(* IEC 61131-3 sources: lacyccom-procedural/src/drive_functions/blocks (part 3) *)

(* ---- LAcycCom_DriveRamToRom.st ---- *)
USING System.Timer;
USING Siemens.Simatic.DistributedIO;

NAMESPACE Simatic.Ax.LAcycCom.Procedural
  TYPE INTERNAL
    LAcycCom_DriveRamToRomStates : SINT (
      FB_IDLE := SINT#0,   // Idle state in FB
      FB_FIRST_CYCLE := SINT#1,   // First cycle state in FB
      FB_ALLOCATE := SINT#2,   // Allocating a buffer element in request buffer DB
      FB_GET_RESOURCE := SINT#3,   // State to check if the communication to the drive object can be established
      FB_BUSY := SINT#4,   // Busy state in FB
      FB_RELEASE := SINT#5,   // State to return the allocated index
      FB_DONE := SINT#6,   // Done state in FB
      FB_ERROR := SINT#7,   // Error state in FB
      FB_BUSY_READ := SINT#8,   // State of configuration drive object data (read parameter r3996)
      FB_BUSY_WriteRecord_READ := SINT#9,   // WriteRecord in busy state
      FB_BUSY_ReadRecord_READ := SINT#10,   // ReadRecord in busy state
      FB_BUSY_WRITE_PARAM_971 := SINT#11,   // State of configuration drive object data (write parameter p971)
      FB_BUSY_WriteRecord_WRITE_PARAM_971 := SINT#12,   // WriteRecord in busy state
      FB_BUSY_ReadRecord_WRITE_PARAM_971 := SINT#13,   // ReadRecord in busy state
      FB_BUSY_WRITE_PARAM_977 := SINT#14,   // State of configuration drive object data (write parameter p977)
      FB_BUSY_WriteRecord_WRITE_PARAM_977 := SINT#15,   // WriteRecord in busy state
      FB_BUSY_ReadRecord_WRITE_PARAM_977 := SINT#16,   // ReadRecord in busy state
      FB_BUSY_CYCLE_TIMER := SINT#17,   // Cyclic OnDelay in busy state
      FB_BUSY_CHECK_PARAM_971 := SINT#18,   // State of configuration drive object data (read parameter r3996)
      FB_BUSY_WriteRecord_CHECK_971 := SINT#19,   // WriteRecord in busy state
      FB_BUSY_ReadRecord_CHECK_971 := SINT#20,   // ReadRecord in busy state
      FB_BUSY_CHECK_PARAM_977 := SINT#21,   // State of configuration drive object data (read parameter p977)
      FB_BUSY_WriteRecord_CHECK_977 := SINT#22,   // WriteRecord in busy state
      FB_BUSY_ReadRecord_CHECK_977 := SINT#23,   // ReadRecord in busy state
      FB_BUSY_CHECK_PROGRESS := SINT#24,   // Check RAM to ROM progress
      FB_BUSY_WAIT := SINT#25   // State when temporary error occurred
    ) := FB_IDLE;
  END_TYPE

  ///------------------------------------------------------------------------------------------
  /// SIEMENS AG
	/// (c)Copyright 2026 All Rights Reserved
	///------------------------------------------------------------------------------------------
	/// Library: LAcycCom
	/// Tested with: S7-1513-1 PN
	/// Engineering: SIMATIC AX
	/// Restrictions: ---
	/// Requirements: S7-1200 / S7-1500
	///               FB LAcycCom_ResourceManager is required
	/// Functionality: Copy RAM to ROM of a specific drive object.
  ///------------------------------------------------------------------------------------------
  FUNCTION_BLOCK LAcycCom_DriveRamToRom
    {S7.Extern = ReadWrite}
    VAR_INPUT
      execute : BOOL;   /// TRUE: Rising edge starts the functionality once
      driveObjectId : INT := -1;   /// Optional: Identification number of the drive object (value <0: driveObjectId is not used, i.e. the corresponding drive object is only addressed via the hardwareId)
      hardwareId : UINT;   /// Hardware identifier of the hardware module
      enableSavingOfWholeDriveSystem : BOOL;   /// TRUE: Enable saving of all parameters of all drive objects of a multi drive system (e.g. S120). Note: parameter p977 must therefore be available at the addressed drive object. If p977 is not available p971 is written, i.e., the setting also works for single drive systems (e.g. G120)
    END_VAR

    {S7.Extern = ReadOnly}
    VAR_OUTPUT
      done : BOOL;   /// TRUE: RAM data successfully written to ROM
      busy : BOOL;   /// TRUE: FB is not finished and new output values can be expected
      error : BOOL;   /// TRUE: Rising edge informs that an error occurred during the execution of the FB
      status : LAcycCom_DriveFunctionStatus := LAcycCom_DriveFunctionStatus#STATUS_NO_CALL;   /// Status identifier
      diagnostics : LAcycCom_typeDriveDiagnostics;   /// Diagnostics structure
    END_VAR

    VAR_IN_OUT
      requestBufferHeader : LAcycCom_typeRequestBufferHeader;   /// Interface for header of request buffer
      requestBuffer : ARRAY[*] OF LAcycCom_typeRequestBufferElement;   /// Interface for request buffer
    END_VAR

    VAR
      _busy : BOOL := FALSE;   /// Static value for output busy
      _done : BOOL := FALSE;   /// Static value for output done
      _error : BOOL := FALSE;   /// Static value for output error
      _executeOld : BOOL := FALSE;   /// Old value of execute for edge detection
      _cmdBusy : BOOL := FALSE;   /// TRUE: Process is not yet complete
      _cmdDone : BOOL := FALSE;   /// TRUE: Data record was transferred
      _cmdError : BOOL := FALSE;   /// TRUE: An error occurred during processing
      _timerStart : BOOL := FALSE;   /// TRUE: Starts OnDelay
      _refNo : BYTE := BYTE#16#00;   /// Reference number of request
      _doId : BYTE := BYTE#16#00;   /// Intern identification number of the drive object
      _status : LAcycCom_DriveFunctionStatus := LAcycCom_DriveFunctionStatus#STATUS_NO_CALL;   /// Static value for output status
      _subfunctionStatus : WORD := WORD#16#0000;   /// Block status or error information
      _withoutResourceManager : BOOL := FALSE;   /// TRUE: No resource manager available; FALSE: Resource manager available
      _stateNumber : SINT := SINT#0;   /// State of the FB when error occurred
      _fbState : SINT := LAcycCom_DriveRamToRomStates#FB_IDLE;   /// States in the function block state machine
      _fbSubState : SINT := LAcycCom_DriveRamToRomStates#FB_BUSY_WriteRecord_WRITE_PARAM_971;   /// States in the function block during processing (busy state)
      _fbSubStateOld : SINT := LAcycCom_DriveRamToRomStates#FB_BUSY_WriteRecord_WRITE_PARAM_971;   /// Previous state when temporary error occurs
      _errorCount : UInt := UINT#0;   /// Error counter of retry request
      _allocatedIndex : INT := 0;   /// Allocated element index in the buffer DB
      _countOfElements : INT := 0;   /// Number of parameters in the dataset
      _firstParameterError : INT := -1;   /// Number of parameter at which the error occurred (-1: no parameter with error)
      _hwId : UINT := UINT#0;   /// Intern hardware identifier of the hardware module
      _warningRetriggering : BOOL;   /// TRUE: Input execute is set during processing
      _dataRecordNo : DINT;   /// Used data record
      _cyclicTimerStart : BOOL;   /// TRUE: Starts the OnDelay
      _parameter : ARRAY[0..NO_OF_PARAMETERS_UPPER_LIM] OF LAcycCom_typeParameter;   /// Parameter dataset
      _parameterRam2Rom : ARRAY[0..0] of LAcycCom_typeParameter;   /// Parameter dataset for write Ram2Rom
      _reqWriteParameterHeader : LAcycCom_typeParameterHeader;   /// Request telegram to change the parameter values
      _reqWriteParameterData : ARRAY[0..LENGTH_WRITE_PARAMETER_TELEGRAM_UPPER_LIM] OF BYTE;   /// List of parameter (max. 16 parameter)
      _reqReadParameterHeader : LAcycCom_typeParameterHeader;   /// Request telegram
      _reqReadParameterAddress : ARRAY[0..NO_OF_PARAMETERS_UPPER_LIM] OF LAcycCom_typeParameterAddress;   /// Parameter data in telegram
      _respParameterHeader : LAcycCom_typeParameterHeader;   /// Response telegram
      _respParameterData : ARRAY[0..LENGTH_READ_PARAMETER_TELEGRAM_UPPER_LIM] OF BYTE;   /// List of parameter (max. 16 parameter)
      _reqReadParameterInit : LAcycCom_typeParameterAddress := ( attribute := BYTE#16#10, elementNo := BYTE#16#01, parameterNo := UINT#0, index := UINT#0 );   /// Initialisation of the parameter dataset
      _instWriteRecord  : WriteRecord;   /// WriteRecord command
      _instReadRecord : ReadRecord;   /// ReadRecord command
      _instOnDelay : OnDelay;   /// OnDelay
    END_VAR

    VAR_TEMP
      tempCmdValid : BOOL;   // TRUE: New data record was received and is valid
      tempIndex : INT;   // Temporary loop index variable
      tempLastQueueElement : INT;   // Last element in queue
      tempPointer : INT;   // Temporary pointer variable
      tempWord : WORD;   // Temporary word variable
      tempUDint : UDINT;   // Temporary udint variable
      tempStatusWord : WORD;   // Temporary status
      tempCmdStatus : DWORD;   // Temporary status of WriteRecord and ReadRecord command
      tempVoidDiagnostics : LAcycCom_typeDriveDiagnostics;   // Temporary empty diagnostics structure
      tempVoidHeader : LAcycCom_typeParameterHeader;   // Temporary empty header structure
      tempRecord : ARRAY[0..239] OF BYTE;   // Temporary record buffer for WriteRecord and ReadRecord instruction
    END_VAR

    VAR CONSTANT
      MAX_ERROR_COUNT : UINT := UINT#40;   // Maximum error counter
      NO_OF_PARAMETERS_UPPER_LIM : INT := 1;   // Maximum count of parameters
      LENGTH_WRITE_PARAMETER_TELEGRAM_UPPER_LIM : INT := 23;   // Maximum length of write telegram in Byte
      LENGTH_READ_PARAMETER_TELEGRAM_UPPER_LIM : INT := 11;   // Maximum length of read telegram in Byte
      ALL_ELEMENTS_OCCUPIED : INT := -1;   // All buffer elements are occupied
      TIMER_ALLOCATION : TIME := T#10S;   // Timer limit for allocating a buffer element
      TIMER_TEMP_ERROR : TIME := T#200MS;   // Waiting time until next system function block call
      TIMER_CYCLIC : TIME := T#500MS;   // Timer interval of checking the result of the Ram to Rom process
      MAX_DRIVE_OBJECT_NO : INT := 254;   // Maximum drive object number limited by SINAMICS p101
    END_VAR

    // Check if FB is triggered
    IF (execute = TRUE) AND (_executeOld = FALSE) AND (_busy = TRUE) THEN
      // Input execute is set during processing
      _status := LAcycCom_DriveFunctionStatus#WARN_EXECUTE_SET_DURING_PROCESSING;
      _warningRetriggering := TRUE;
      _executeOld := execute;

    ELSIF (execute = TRUE) AND (_executeOld = FALSE) THEN
      // First call
      // Initialisation
      _done := FALSE;
      _error := FALSE;
      //_status := LAcycCom_DriveFunctionStatus#STATUS_FIRST_CALL;
      _allocatedIndex := 0;
      _hwId := UINT#0;
      _subfunctionStatus := WORD#16#0;
      _doId := BYTE#0;
      _dataRecordNo := 0;
      _stateNumber := SINT#0;
      _firstParameterError := -1;
      _cmdBusy := FALSE;
      _cmdDone := FALSE;
      _cmdError := FALSE;
      _errorCount := UINT#0;
      _countOfElements := 0;
      _warningRetriggering := FALSE;
      _fBSubState := LAcycCom_DriveRamToRomStates#FB_BUSY_READ;
      _fBState := LAcycCom_DriveRamToRomStates#FB_FIRST_CYCLE;

      // Initialize functionality after triggering FB, e.g. reset of values
      //-----------------------------------------------------------------------------------
      _instOnDelay(signal := FALSE,
              duration := TIMER_ALLOCATION);

      // Functionality is busy
      _busy := TRUE;

      // Reset other outputs
      _error := FALSE;
      //_status := LAcycCom_DriveFunctionStatus#STATUS_FIRST_CALL;

      busy := _busy;
      error := _error;
      _executeOld := execute;
      RETURN;

      // FB is currently inactive
    ELSIF (execute = FALSE) AND (_busy = FALSE) AND
        (_error = TRUE OR _done = TRUE)
    THEN
      _error := FALSE;
      _busy := FALSE;
      _done := FALSE;
      _fBState := LAcycCom_DriveRamToRomStates#FB_IDLE;

      // Write outputs
      _status := LAcycCom_DriveFunctionStatus#STATUS_NO_CALL;
      busy := _busy;
      done := _done;
      error := _error;

      _executeOld := execute;
      RETURN;

      // FB is currently executed and not finished
    ELSIF _busy = TRUE THEN
      _executeOld := execute;

      // FB finished request
    ELSE
      _executeOld := execute;
      RETURN; //Wait for start of functionality
    END_IF;
    //----------------------------------------------------------------------------------------------

    IF (_busy = TRUE) AND (_error = FALSE) THEN  // Functionality running
        CASE _fBState OF
            LAcycCom_typeDriveActDeactStates#FB_FIRST_CYCLE:  // First cycle state

            // Clearing the sending reading buffer
            _reqReadParameterHeader := tempVoidHeader;
            _reqReadParameterAddress[0] := _reqReadParameterInit;

            // Clearing the sending write buffer
            _reqWriteParameterHeader := tempVoidHeader;
            FOR tempIndex := 0 TO LENGTH_WRITE_PARAMETER_TELEGRAM_UPPER_LIM DO
            _reqWriteParameterData[tempIndex] := BYTE#16#00;
            END_FOR;

            // Clearing the receive buffer
            _respParameterHeader := tempVoidHeader;
            FOR tempIndex := 0 TO LENGTH_READ_PARAMETER_TELEGRAM_UPPER_LIM DO
            _respParameterData[tempIndex] := BYTE#16#00;
            END_FOR;

            // Initialization after start
            IF driveObjectId < 0 THEN // V1.5
            _dataRecordNo := 16#B02E; // Base Mode Parameter Access local; doId not relevant
            _doId := BYTE#0;

            ELSIF (driveObjectId <= MAX_DRIVE_OBJECT_NO)
            AND (driveObjectId <> 0)
            THEN // V1.5.2
            _dataRecordNo := 47; // Data record 47; Base Mode Parameter Access global
            _doId := TO_BYTE(driveObjectId);

            ELSE // V1.5.2
            // Wrong drive object ID at input
            _error := TRUE;
            _stateNumber := _fBState;
            _status := LAcycCom_DriveFunctionStatus#ERR_INVALID_DRIVE_OBJECT_ID;
            _fBState := LAcycCom_typeDriveActDeactStates#FB_ERROR;
            END_IF;

            _hwId := hardwareId;
            diagnostics := tempVoidDiagnostics;
            diagnostics.driveObjectId := TO_SINT(_doId);
            diagnostics.hardwareId := _hwId;
            diagnostics.parameterCount := 2;
            _countOfElements := 2;
            diagnostics.firstParameterError := _firstParameterError; // V1.3.2
            diagnostics.errorValue := BYTE#16#FF; // V1.3.2

            _parameter[0].parameterNo := UINT#0;
            _parameter[1].parameterNo := UINT#0;
            _parameterRam2Rom[0].parameterNo := UINT#0; // V1.3.3

            _parameter[0].index := UINT#0;
            _parameter[1].index := UINT#0;
            _parameterRam2Rom[0].index := UINT#0;

            _parameter[0].realValue := REAL#0.0;
            _parameter[1].realValue := REAL#0.0;
            _parameterRam2Rom[0].realValue := REAL#0.0;

            _parameter[0].format := BYTE#16#00;
            _parameter[1].format := BYTE#16#00;
            _parameterRam2Rom[0].format := BYTE#16#00;

            _parameter[0].errorValue := BYTE#16#00;
            _parameter[1].errorValue := BYTE#16#00;
            _parameterRam2Rom[0].errorValue := BYTE#16#00;

            // Next state is depending on the FB mode
            IF (_withoutResourceManager = FALSE) AND (_error = FALSE) THEN
            _status := LAcycCom_DriveFunctionStatus#STATUS_ALLOCATE;
            _fBState := LAcycCom_typeDriveActDeactStates#FB_ALLOCATE;

            ELSIF (_withoutResourceManager = TRUE) AND (_error = FALSE) THEN
            _status := LAcycCom_DriveFunctionStatus#STATUS_BUSY;
            _fBState := LAcycCom_typeDriveActDeactStates#FB_BUSY;
            _fBSubState := LAcycCom_DriveRamToRomStates#FB_BUSY_READ;
            END_IF;

            LAcycCom_typeDriveActDeactStates#FB_ALLOCATE:
            // Allocation of a buffer element
            IF (requestBufferHeader.lockBuffer = FALSE) AND (requestBufferHeader.nextFreeElement >= requestBufferHeader.bufferLowerBound) AND (requestBufferHeader.nextFreeElement <= requestBufferHeader.bufferUpperBound) THEN
            requestBufferHeader.lockBuffer := TRUE;
            _allocatedIndex := requestBufferHeader.nextFreeElement;
            requestBuffer[_allocatedIndex].state := BYTE#16#00;
            requestBuffer[_allocatedIndex].state.%X0 := TRUE;
            requestBuffer[_allocatedIndex].hardwareId := _hwId;
            requestBuffer[_allocatedIndex].queueElementNext := -1;
            _timerStart := FALSE;
            _status := LAcycCom_DriveFunctionStatus#STATUS_GET_RESOURCE;
            _fBState := LAcycCom_typeDriveActDeactStates#FB_GET_RESOURCE;

            // Build up queue
            IF (requestBufferHeader.firstQueueElement >= 0) THEN
                // Find last queue element
                tempIndex := requestBufferHeader.firstQueueElement;
                WHILE (tempIndex >= 0) DO
                tempLastQueueElement := tempIndex;
                tempIndex := requestBuffer[tempIndex].queueElementNext;
                END_WHILE;

                // Insert into list after last element
                requestBuffer[tempLastQueueElement].queueElementNext := _allocatedIndex;
                requestBuffer[_allocatedIndex].queueElementPrevious := tempLastQueueElement;

            ELSE
                // Element is first element in queue
                requestBufferHeader.firstQueueElement := _allocatedIndex;
                requestBuffer[_allocatedIndex].queueElementPrevious := -1;
            END_IF;

            // Searching for the next free buffer element
            FOR tempIndex := requestBufferHeader.bufferLowerBound TO TO_INT(requestBufferHeader.bufferUpperBound) DO
                IF (requestBuffer[tempIndex].state.%X0 = FALSE) THEN
                requestBufferHeader.nextFreeElement := tempIndex;
                EXIT;
                END_IF;

                // All buffer elements are occupied
                IF (tempIndex = requestBufferHeader.bufferUpperBound) THEN
                requestBufferHeader.nextFreeElement := ALL_ELEMENTS_OCCUPIED;
                END_IF;
            END_FOR;

            requestBufferHeader.lockBuffer := FALSE;

            ELSIF (_instOnDelay.output = TRUE) THEN
            _error := TRUE;
            _stateNumber := _fBState;
            _status := LAcycCom_DriveFunctionStatus#ERR_ALLOCATION_TIME;
            _fBState := LAcycCom_typeDriveActDeactStates#FB_ERROR;

            ELSE
            ; // Waiting until lockbit is reset and a buffer element is available
            END_IF; // (#buffer.lockBuffer = FALSE) AND (#buffer.actualWriteIndex >= 0)

            _instOnDelay(signal := _timerStart,
                    duration := TIMER_ALLOCATION);

            _timerStart := TRUE;
            IF (_instOnDelay.output = TRUE) THEN
            _timerStart := FALSE;
            END_IF;

            LAcycCom_typeDriveActDeactStates#FB_GET_RESOURCE:

            // Check buffer index for correctness
            IF (_allocatedIndex < requestBufferHeader.bufferLowerBound) OR (_allocatedIndex > requestBufferHeader.bufferUpperBound) THEN
            _error := TRUE;
            _stateNumber := _fBState;
            _status := LAcycCom_DriveFunctionStatus#ERR_INVALID_BUF_INDEX;
            _fBState := LAcycCom_typeDriveActDeactStates#FB_ERROR;

            ELSE
            IF (requestBuffer[_allocatedIndex].state.%X0 = FALSE) OR
                (requestBuffer[_allocatedIndex].state.%X3 = TRUE)
            THEN
                // Request was rejected by buffer manager
                _error := TRUE;
                _stateNumber := _fBState;
                _status := LAcycCom_DriveFunctionStatus#ERR_REQUEST_REJECTED;
                _fBState := LAcycCom_typeDriveActDeactStates#FB_ERROR;

            ELSIF (requestBuffer[_allocatedIndex].state.%X2 = TRUE) THEN
                // Request already released
                _error := TRUE;
                _stateNumber := _fBState;
                _status := LAcycCom_DriveFunctionStatus#ERR_RESOURCE_RELEASED;
                _fBState := LAcycCom_typeDriveActDeactStates#FB_ERROR;

            ELSIF (requestBuffer[_allocatedIndex].state.%X1 = TRUE) THEN
                // Element is enabled
                _status := LAcycCom_DriveFunctionStatus#STATUS_BUSY;
                _fBState := LAcycCom_typeDriveActDeactStates#FB_BUSY;
                _fBSubState := LAcycCom_DriveRamToRomStates#FB_BUSY_READ;

            ELSE
                // Element not enabled yet
                //
                _status := LAcycCom_DriveFunctionStatus#STATUS_GET_RESOURCE;
            END_IF;

            END_IF;

            LAcycCom_typeDriveActDeactStates#FB_BUSY:

            IF ((requestBuffer[_allocatedIndex].state.%X1 = TRUE) AND (_withoutResourceManager = FALSE) AND ((requestBuffer[_allocatedIndex].state.%X3 = FALSE))) OR
            (_withoutResourceManager = TRUE)
            THEN

            CASE _fBSubState OF

                LAcycCom_DriveRamToRomStates#FB_BUSY_READ:
                // Creating header data
                _refNo := TO_BYTE(TO_SINT(_refNo) + 1);
                _reqReadParameterHeader.refNo := _refNo; // Telegram reference number
                _reqReadParameterHeader.reqId := BYTE#16#01;  // 0x01 = request parameters
                _reqReadParameterHeader.doId := _doId;  // Drive object identification number
                _reqReadParameterHeader.parameterNo := TO_BYTE(_countOfElements);  // Count of parameters

                // Copying the dataset into a static variable (depending on the used PLC data type)
                _parameter[0].index := UINT#0;
                _parameter[0].parameterNo := UINT#971; // Save drive object parameters
                _parameter[0].format := TO_BYTE(LAcycCom_DriveValueFormats#FORMAT_UNSIGNED_16);
                _parameter[1].index := UINT#0;
                _parameter[1].parameterNo := UINT#977; // Save all parameters
                _parameter[1].format := TO_BYTE(LAcycCom_DriveValueFormats#FORMAT_UNSIGNED_16);

                _reqReadParameterAddress[0].attribute := BYTE#16#10; // Attribute of parameters (0x10=Value, 0x30=Text)
                _reqReadParameterAddress[0].elementNo := BYTE#16#01; // No. of elements (for single elements=1)

                _reqReadParameterAddress[1].attribute := BYTE#16#10; // Attribute of parameters (0x10=Value, 0x30=Text)
                _reqReadParameterAddress[1].elementNo := BYTE#16#01; // No. of elements (for single elements=1)

                // Parameter number
                _reqReadParameterAddress[0].parameterNo := _parameter[0].parameterNo;
                _reqReadParameterAddress[1].parameterNo := _parameter[1].parameterNo;

                // Subindex of parameter
                _reqReadParameterAddress[0].index := _parameter[0].index;
                _reqReadParameterAddress[1].index := _parameter[1].index;

                _status := LAcycCom_DriveFunctionStatus#STATUS_BUSY;
                _fBState := LAcycCom_typeDriveActDeactStates#FB_BUSY;
                _fBSubState := LAcycCom_DriveRamToRomStates#FB_BUSY_WriteRecord_READ;

                LAcycCom_DriveRamToRomStates#FB_BUSY_WRITE_PARAM_971, LAcycCom_DriveRamToRomStates#FB_BUSY_WRITE_PARAM_977:

                // Initialize diagnostics and count of elements
                diagnostics.parameterCount := 1;
                _countOfElements := 1;

                // Clearing the receive buffer V1.3.3
                _respParameterHeader := tempVoidHeader;
                FOR tempIndex := 0 TO LENGTH_READ_PARAMETER_TELEGRAM_UPPER_LIM DO
                    _respParameterData[tempIndex] := BYTE#16#00;
                END_FOR;

                // Creating header data
                _refNo := TO_BYTE(TO_SINT(_refNo) + 1);
                _reqWriteParameterHeader.refNo := _refNo; // Telegram reference number
                _reqWriteParameterHeader.reqId := BYTE#16#02;  // 0x02 = change parameters
                _reqWriteParameterHeader.doId := _doId;  // Drive object identification number of CU
                _reqWriteParameterHeader.parameterNo := TO_BYTE(_countOfElements);  // Count of parameters

                // Copying the dataset into a static variable
                _parameterRam2Rom[0].index := UINT#0;
                IF (_fBSubState = LAcycCom_DriveRamToRomStates#FB_BUSY_WRITE_PARAM_971) THEN // V1.3.3
                    _parameterRam2Rom[0].parameterNo := UINT#971; // Save drive object parameters
                    _fBSubState := LAcycCom_DriveRamToRomStates#FB_BUSY_WriteRecord_WRITE_PARAM_971;
                ELSE
                    _parameterRam2Rom[0].parameterNo := UINT#977; // Save all parameters
                    _fBSubState := LAcycCom_DriveRamToRomStates#FB_BUSY_WriteRecord_WRITE_PARAM_977;
                END_IF;

                _parameterRam2Rom[0].format := TO_BYTE(LAcycCom_DriveValueFormats#FORMAT_UNSIGNED_16);
                _parameterRam2Rom[0].realValue := REAL#1.0;

                // Write parameter address
                _reqWriteParameterData[0] := BYTE#16#10; // Attribute of parameters (0x10=Value, 0x30=Text)
                _reqWriteParameterData[1] := BYTE#16#01; // No. of elements (for single elements=1)

                // Parameter number
                _reqWriteParameterData[2] := _parameterRam2Rom[0].parameterNo.%B1;
                _reqWriteParameterData[3] := _parameterRam2Rom[0].parameterNo.%B0;

                // Subindex of parameter
                _reqWriteParameterData[4] := _parameterRam2Rom[0].index.%B1;
                _reqWriteParameterData[5] := _parameterRam2Rom[0].index.%B0;

                _reqWriteParameterData[6] := _parameterRam2Rom[0].format; // Format of parameter
                _reqWriteParameterData[7] := BYTE#16#01; // Count of values

                // Parameter value (= 1.0)
                _reqWriteParameterData[8] := BYTE#16#00;
                _reqWriteParameterData[9] := BYTE#16#01;

                _status := LAcycCom_DriveFunctionStatus#STATUS_BUSY;
                _fBState := LAcycCom_typeDriveActDeactStates#FB_BUSY;

                LAcycCom_DriveRamToRomStates#FB_BUSY_CYCLE_TIMER:

                // Start cyclic timer
                _instOnDelay(signal := _cyclicTimerStart,
                              duration := TIMER_CYCLIC);

                _cyclicTimerStart := TRUE;
                IF (_instOnDelay.output = TRUE) THEN
                    _cyclicTimerStart := FALSE;
                    _fBSubState := _fBSubStateOld; // V1.3.3
                END_IF;

                LAcycCom_DriveRamToRomStates#FB_BUSY_CHECK_PARAM_971, LAcycCom_DriveRamToRomStates#FB_BUSY_CHECK_PARAM_977:

                // Clearing the receive buffer V1.3.3
                _respParameterHeader := tempVoidHeader;
                FOR tempIndex := 0 TO LENGTH_READ_PARAMETER_TELEGRAM_UPPER_LIM DO
                    _respParameterData[tempIndex] := BYTE#16#00;
                END_FOR;

                // Creating header data
                _refNo := TO_BYTE(TO_SINT(_refNo) + 1);
                _reqReadParameterHeader.refNo := _refNo; // Telegram reference number
                _reqReadParameterHeader.reqId := BYTE#16#01;  // 0x01 = request parameters
                _reqReadParameterHeader.doId := _doId;  // Drive object identification number of CU
                _reqReadParameterHeader.parameterNo := TO_BYTE(_countOfElements);  // Count of parameters

                IF _fBSubState = LAcycCom_DriveRamToRomStates#FB_BUSY_CHECK_PARAM_971 THEN // V1.3.3
                    _parameterRam2Rom[0].parameterNo := UINT#971; // Save drive object parameters
                    _fBSubState := LAcycCom_DriveRamToRomStates#FB_BUSY_WriteRecord_CHECK_971;

                ELSE
                    _parameterRam2Rom[0].parameterNo := UINT#977; // Save all parameters
                    _fBSubState := LAcycCom_DriveRamToRomStates#FB_BUSY_WriteRecord_CHECK_977;
                END_IF;

                _parameterRam2Rom[0].format := TO_BYTE(LAcycCom_DriveValueFormats#FORMAT_UNSIGNED_16);

                _status := LAcycCom_DriveFunctionStatus#STATUS_BUSY;
                _fBState := LAcycCom_typeDriveActDeactStates#FB_BUSY;

                // Copying the dataset into a static variable (depending on the used PLC data type)
                _parameterRam2Rom[0].index := UINT#0;

                _reqReadParameterAddress[0].attribute := BYTE#16#10; // Attribute of parameters (0x10=Value, 0x30=Text)
                _reqReadParameterAddress[0].elementNo := BYTE#16#01; // No. of elements (for single elements=1)

                // Parameter number
                _reqReadParameterAddress[0].parameterNo := _parameterRam2Rom[0].parameterNo;

                // Subindex of parameter
                _reqReadParameterAddress[0].index := _parameterRam2Rom[0].index;

                LAcycCom_DriveRamToRomStates#FB_BUSY_CHECK_PROGRESS:

                IF (_parameterRam2Rom[0].realValue = REAL#0.0) // Ram2Rom is completed
                THEN

                    // Next state is depending on the FB mode
                    IF (_withoutResourceManager = FALSE) AND (_error = FALSE) THEN
                    _status := LAcycCom_DriveFunctionStatus#STATUS_RELEASE;
                    _fBState := LAcycCom_typeDriveActDeactStates#FB_RELEASE;

                    ELSIF (_withoutResourceManager = TRUE) AND (_error = FALSE) THEN
                    _status := LAcycCom_DriveFunctionStatus#STATUS_EXECUTION_FINISHED;
                    _fBState := LAcycCom_typeDriveActDeactStates#FB_DONE;
                    END_IF; // _mode = #MODE_WITH_BUFFER_MANAGER

                ELSE
                    _status := LAcycCom_DriveFunctionStatus#STATUS_BUSY;
                    _fBSubState := LAcycCom_DriveRamToRomStates#FB_BUSY_CYCLE_TIMER;
                END_IF;

                // Writing the dataset configuration into the drive object
                LAcycCom_DriveRamToRomStates#FB_BUSY_WriteRecord_READ, LAcycCom_DriveRamToRomStates#FB_BUSY_WriteRecord_WRITE_PARAM_971, LAcycCom_DriveRamToRomStates#FB_BUSY_WriteRecord_WRITE_PARAM_977, LAcycCom_DriveRamToRomStates#FB_BUSY_WriteRecord_CHECK_971, LAcycCom_DriveRamToRomStates#FB_BUSY_WriteRecord_CHECK_977:

                IF (_cmdBusy = FALSE) THEN
                    // Resets WriteRecord command
                    _instWriteRecord(request := FALSE,
                        record := tempRecord);

                END_IF; // _cmdBusy = FALSE

                IF ((_fBSubState = LAcycCom_DriveRamToRomStates#FB_BUSY_WriteRecord_WRITE_PARAM_971) OR (_fBSubState = LAcycCom_DriveRamToRomStates#FB_BUSY_WriteRecord_WRITE_PARAM_977)) AND (_error = FALSE) THEN
                    SerializeParamWrite(_reqWriteParameterHeader, _reqWriteParameterData, tempRecord);
                    // WriteRecord command
                    _instWriteRecord(request := TRUE,                                                     // Transfer data record
                                      hardwareId := _hwId,                                                 // ID number of the hardware component
                                      index := _dataRecordNo,                                      // Data record number
                                      length := UINT#0,                                                        // Maximum length of the data record to be transferred in bytes
                                      done => _cmdDone,                                            // Data record was transferred
                                      busy => _cmdBusy,                                            // The writing process is not yet complete
                                      error => _cmdError,                                          // An error occurred during the writing process
                                      status => tempCmdStatus,                                        // Status[1] = Error => Status[2] Error Decode + Status[3] Error Code
                                      record := tempRecord);                               // Data record

                ELSIF ((_fBSubState = LAcycCom_DriveRamToRomStates#FB_BUSY_WriteRecord_CHECK_971) OR (_fBSubState = LAcycCom_DriveRamToRomStates#FB_BUSY_WriteRecord_READ) OR (_fBSubState = LAcycCom_DriveRamToRomStates#FB_BUSY_WriteRecord_CHECK_977))
                    AND (_error = FALSE)
                THEN
                    SerializeParamAddress(_reqReadParameterHeader, _reqReadParameterAddress, tempRecord);
                    // WriteRecord command
                    _instWriteRecord(request := TRUE,                                                     // Transfer data record
                                      hardwareId := _hwId,                                                 // ID number of the hardware component
                                      index := _dataRecordNo,                                      // Data record number
                                      length := UINT#0,                                                        // Maximum length of the data record to be transferred in bytes
                                      done => _cmdDone,                                            // Data record was transferred
                                      busy => _cmdBusy,                                            // The writing process is not yet complete
                                      error => _cmdError,                                          // An error occurred during the writing process
                                      status => tempCmdStatus,                                        // Status[1] = Error => Status[2] Error Decode + Status[3] Error Code
                                      record := tempRecord);                                // Data record
                END_IF;

                // Error occurred
                IF (_cmdError = TRUE) AND (_error = FALSE) THEN
                    tempStatusWord.%B0 := tempCmdStatus.%B1;
                    tempStatusWord.%B1 := tempCmdStatus.%B2;

                    // Temporary command status (80A1, 80A7, 80B5, 80C0, 80C1, 80C2, 80C3 or 80C4) are valid and retry command
                    IF (tempStatusWord = WORD#16#80A1) OR  // Negative acknowledgment when writing to the module
                    (tempStatusWord = WORD#16#80A7) OR   // DP slave or module is occupied (temporary error)
                    (tempStatusWord = WORD#16#80B5) OR   // DP slave or module not ready
                    (tempStatusWord = WORD#16#80C0) OR   // The data can only be written when the CPU is in STOP mode. Note: this means that writing by the user program is not possible. You can only write the data online with PG/PC.
                    (tempStatusWord = WORD#16#80C1) OR   // The data of the previous write job on the module for the same data record have not yet been processed by the module.
                    (tempStatusWord = WORD#16#80C2) OR   // The module is currently processing the maximum possible number of jobs for a CPU.
                    (tempStatusWord = WORD#16#80C3) OR   // The required operating resources are currently occupied.
                    (tempStatusWord = WORD#16#80C4) THEN // Internal temporary error. Job could not be executed. Repeat the job. If this error occurs often, check your installation for sources of electrical interference.

                    IF (_errorCount >= MAX_ERROR_COUNT) THEN
                        _error := TRUE;
                        _stateNumber := _fBSubState;
                        _subfunctionStatus := tempStatusWord;
                        _status := LAcycCom_DriveFunctionStatus#ERR_WRITERECORD_TEMP_COUNTER;
                        _fBState := LAcycCom_typeDriveActDeactStates#FB_ERROR;

                    ELSE
                        _errorCount := _errorCount + UINT#1;  // Increment internal error counter
                        _fBSubStateOld := _fBSubState; // // V1.3.3
                        _fBSubState := LAcycCom_DriveRamToRomStates#FB_BUSY_WAIT;
                    END_IF;

                    ELSIF (_fBSubState = LAcycCom_DriveRamToRomStates#FB_BUSY_WriteRecord_CHECK_971) OR (_fBSubState = LAcycCom_DriveRamToRomStates#FB_BUSY_WriteRecord_CHECK_977) THEN // V1.3.3
                    _error := TRUE;
                    _stateNumber := _fBSubState;
                    _subfunctionStatus := tempStatusWord;
                    _status := LAcycCom_DriveFunctionStatus#ERR_MISSING_CONFIRMATION;
                    _fBState := LAcycCom_typeDriveActDeactStates#FB_ERROR;

                    ELSE
                    _error := TRUE;
                    _stateNumber := _fBSubState;
                    _subfunctionStatus := tempStatusWord;
                    _status := LAcycCom_DriveFunctionStatus#ERR_WRITERECORD;
                    _fBState := LAcycCom_typeDriveActDeactStates#FB_ERROR;
                    END_IF;

                ELSIF (_cmdDone = TRUE) AND (_error = FALSE) AND (_fBSubState = LAcycCom_DriveRamToRomStates#FB_BUSY_WriteRecord_READ) THEN  // Processing completed without errors
                    _errorCount := UINT#0;  // V1.5.1 Reset error counter
                    _fBSubState := LAcycCom_DriveRamToRomStates#FB_BUSY_ReadRecord_READ; // WriteRecord completed and continue with ReadRecord

                ELSIF (_cmdDone = TRUE) AND (_error = FALSE) AND (_fBSubState = LAcycCom_DriveRamToRomStates#FB_BUSY_WriteRecord_WRITE_PARAM_971) THEN  // Processing completed without errors
                    _errorCount := UINT#0;  // V1.5.1 Reset error counter
                    _fBSubState := LAcycCom_DriveRamToRomStates#FB_BUSY_ReadRecord_WRITE_PARAM_971; // WriteRecord completed and continue with ReadRecord

                ELSIF (_cmdDone = TRUE) AND (_error = FALSE) AND (_fBSubState = LAcycCom_DriveRamToRomStates#FB_BUSY_WriteRecord_CHECK_971) THEN  // Processing completed without errors
                    _errorCount := UINT#0;  // V1.5.1 Reset error counter
                    _fBSubState := LAcycCom_DriveRamToRomStates#FB_BUSY_ReadRecord_CHECK_971; // WriteRecord completed and continue with ReadRecord

                ELSIF (_cmdDone = TRUE) AND (_error = FALSE) AND (_fBSubState = LAcycCom_DriveRamToRomStates#FB_BUSY_WriteRecord_WRITE_PARAM_977) THEN  // Processing completed without errors
                    _errorCount := UINT#0;  // V1.5.1 Reset error counter
                    _fBSubState := LAcycCom_DriveRamToRomStates#FB_BUSY_ReadRecord_WRITE_PARAM_977; // WriteRecord completed and continue with ReadRecord

                ELSIF (_cmdDone = TRUE) AND (_error = FALSE) AND (_fBSubState = LAcycCom_DriveRamToRomStates#FB_BUSY_WriteRecord_CHECK_977) THEN  // Processing completed without errors
                    _errorCount := UINT#0;  // V1.5.1 Reset error counter
                    _fBSubState := LAcycCom_DriveRamToRomStates#FB_BUSY_ReadRecord_CHECK_977; // WriteRecord completed and continue with ReadRecord

                END_IF; // _cmdError = TRUE

                // Reading the values from the drive object
                LAcycCom_DriveRamToRomStates#FB_BUSY_ReadRecord_READ, LAcycCom_DriveRamToRomStates#FB_BUSY_ReadRecord_WRITE_PARAM_971, LAcycCom_DriveRamToRomStates#FB_BUSY_ReadRecord_WRITE_PARAM_977, LAcycCom_DriveRamToRomStates#FB_BUSY_ReadRecord_CHECK_971, LAcycCom_DriveRamToRomStates#FB_BUSY_ReadRecord_CHECK_977:
                // Resets ReadRecord command
                IF (_cmdBusy = FALSE) THEN
                    _instReadRecord(request := FALSE,
                        record := tempRecord);
                END_IF;

                _instReadRecord(request := TRUE,                                                    // Transfer data record
                                hardwareID := _hwId,                                        // ID number of the hardware component
                                index := _dataRecordNo,                                     // Data record number
                                maxLength := UINT#0,                                            // Maximum length in bytes of the data record information to be read
                                record := tempRecord,                                          // New data record was received and is valid
                                valid => tempCmdValid,                                      // The reading process is not yet complete
                                busy => _cmdBusy,                                           // An error occurred during the reading process
                                error => _cmdError,                                            // Status[1] = Error => Status[2] Error Decode + Status[3] Error Code
                                status => tempCmdStatus);                                   // Destination area for the data record read

                tempUDint := DeserializeParamResponse(header => _respParameterHeader, response => _respParameterData, buffer := tempRecord);

                IF tempUDint > UDINT#0 THEN
                  // Error occurred
                  IF (_cmdError = TRUE) THEN
                      // Get the error information from the status information
                      tempStatusWord.%B0 := tempCmdStatus.%B1;
                      tempStatusWord.%B1 := tempCmdStatus.%B2;

                      // Temporary command status (80A0, 80A7, 80B5, 80C0, 80C1, 80C2, 80C3 or 80C4) are valid and retry command
                      IF (tempStatusWord = WORD#16#80A0) OR  // Negative acknowledgment when reading the module
                      (tempStatusWord = WORD#16#80A7) OR   // DP slave or module is occupied (temporary error)
                      (tempStatusWord = WORD#16#80B5) OR   // DP slave or module not ready
                      (tempStatusWord = WORD#16#80C0) OR   // The data can only be written when the CPU is in STOP mode. Note: this means that writing by the user program is not possible. You can only write the data online with PG/PC.
                      (tempStatusWord = WORD#16#80C1) OR   // The data of the previous write job on the module for the same data record have not yet been processed by the module.
                      (tempStatusWord = WORD#16#80C2) OR   // The module is currently processing the maximum possible number of jobs for a CPU.
                      (tempStatusWord = WORD#16#80C3) OR   // The required operating resources are currently occupied.
                      (tempStatusWord = WORD#16#80C4) THEN // Internal temporary error. Job could not be executed. Repeat the job. If this error occurs often, check your installation for sources of electrical interference.

                      IF (_errorCount >= MAX_ERROR_COUNT) THEN
                          _error := TRUE;
                          _stateNumber := _fBSubState;
                          _subfunctionStatus := tempStatusWord;
                          _status := LAcycCom_DriveFunctionStatus#ERR_READRECORD_TEMP_COUNTER;
                          _fBState := LAcycCom_typeDriveActDeactStates#FB_ERROR;

                      ELSE
                          _errorCount := _errorCount + UINT#1;  // Increment internal error counter
                          _fBSubStateOld := _fBSubState;
                          // V1.3.2. If error 80A0 then should be retry with WriteRecord command
                          IF (tempStatusWord = WORD#16#80A0) AND _fBSubState = LAcycCom_DriveRamToRomStates#FB_BUSY_ReadRecord_CHECK_971 THEN
                          _fBSubStateOld := LAcycCom_DriveRamToRomStates#FB_BUSY_WriteRecord_CHECK_971;
                          ELSIF (tempStatusWord = WORD#16#80A0) AND _fBSubState = LAcycCom_DriveRamToRomStates#FB_BUSY_ReadRecord_WRITE_PARAM_971 THEN
                          _fBSubStateOld := LAcycCom_DriveRamToRomStates#FB_BUSY_WriteRecord_WRITE_PARAM_971;
                          ELSIF (tempStatusWord = WORD#16#80A0) AND _fBSubState = LAcycCom_DriveRamToRomStates#FB_BUSY_ReadRecord_READ THEN
                          _fBSubStateOld := LAcycCom_DriveRamToRomStates#FB_BUSY_WriteRecord_READ;
                          ELSIF (tempStatusWord = WORD#16#80A0) AND _fBSubState = LAcycCom_DriveRamToRomStates#FB_BUSY_ReadRecord_CHECK_977 THEN
                          _fBSubStateOld := LAcycCom_DriveRamToRomStates#FB_BUSY_WriteRecord_CHECK_977;
                          ELSIF (tempStatusWord = WORD#16#80A0) AND _fBSubState = LAcycCom_DriveRamToRomStates#FB_BUSY_ReadRecord_WRITE_PARAM_977 THEN
                          _fBSubStateOld := LAcycCom_DriveRamToRomStates#FB_BUSY_WriteRecord_WRITE_PARAM_977;
                          END_IF;
                          _fBSubState := LAcycCom_DriveRamToRomStates#FB_BUSY_WAIT;
                      END_IF; // _errorCount >= #MAX_ERROR_COUNT

                      ELSIF (_fBSubState = LAcycCom_DriveRamToRomStates#FB_BUSY_ReadRecord_CHECK_971) OR (_fBSubState = LAcycCom_DriveRamToRomStates#FB_BUSY_ReadRecord_CHECK_977) THEN // V1.3.3
                      _error := TRUE;
                      _stateNumber := _fBSubState;
                      _subfunctionStatus := tempStatusWord;
                      _status := LAcycCom_DriveFunctionStatus#ERR_MISSING_CONFIRMATION;
                      _fBState := LAcycCom_typeDriveActDeactStates#FB_ERROR;

                      ELSE
                      _error := TRUE;
                      _stateNumber := _fBSubState;
                      _subfunctionStatus := tempStatusWord;
                      _status := LAcycCom_DriveFunctionStatus#ERR_READRECORD;
                      _fBState := LAcycCom_typeDriveActDeactStates#FB_ERROR;
                      END_IF;

                      // Error : Reference number of the request does not match with the response reference number
                  ELSIF (_cmdBusy = FALSE) AND
                      (_refNo <> _respParameterHeader.refNo) AND
                      (tempCmdValid = TRUE) THEN

                      _error := TRUE;
                      _stateNumber := _fBSubState;
                      _status := LAcycCom_DriveFunctionStatus#ERR_REFERENCE_NO;
                      _fBState := LAcycCom_typeDriveActDeactStates#FB_ERROR;

                      // Error : Wrong response from the drive object (reqId: 16#01 - reading parameter successful; 16#81: reading parameter finished with error)
                  ELSIF NOT (_respParameterHeader.reqId = BYTE#16#81 OR _respParameterHeader.reqId = BYTE#16#01 OR _respParameterHeader.reqId = BYTE#16#02 OR _respParameterHeader.reqId = BYTE#16#82) AND
                      (_cmdBusy = FALSE) AND
                      (tempCmdValid = TRUE) THEN
                      _error := TRUE;
                      _stateNumber := _fBSubState;
                      _status := LAcycCom_DriveFunctionStatus#ERR_RESPONSE_ID;
                      _fBState := LAcycCom_typeDriveActDeactStates#FB_ERROR;

                      // Error : The received number of parameters does not match with the requested number of parameters
                  ELSIF (_cmdBusy = FALSE) AND
                      (TO_INT(_respParameterHeader.parameterNo) <> _countOfElements) AND
                      (tempCmdValid = TRUE) THEN

                      _error := TRUE;
                      _stateNumber := _fBSubState;
                      _status := LAcycCom_DriveFunctionStatus#ERR_PARAMETER_NO;
                      _fBState := LAcycCom_typeDriveActDeactStates#FB_ERROR;

                      // Error : The drive object does not match with the responsed DO
                  ELSIF (_cmdBusy = FALSE) AND
                      (_respParameterHeader.doId <> _doId) AND
                      (tempCmdValid = TRUE) THEN

                      _error := TRUE;
                      _stateNumber := _fBSubState;
                      _status := LAcycCom_DriveFunctionStatus#ERR_DRIVE_OBJECT_NO;
                      _fBState := LAcycCom_typeDriveActDeactStates#FB_ERROR;

                      // No error occurred during reading parameters
                  ELSIF (_cmdBusy = FALSE) AND (tempCmdValid = TRUE) AND (_error = FALSE) THEN
                      // Analyse of the response buffer

                      IF (_fBSubState = LAcycCom_DriveRamToRomStates#FB_BUSY_ReadRecord_READ) THEN // V1.3.3
                      // If p971 is available then write p971
                      // otherwise write p977 (e.g. drive S210)

                      // Analyse of the response buffer
                      tempPointer := 0;
                      FOR tempIndex := 0 TO NO_OF_PARAMETERS_UPPER_LIM DO
                          _parameter[tempIndex].format := _respParameterData[tempPointer];  // Format of the parameter
                          // Format = Error
                          IF (((TO_SINT(_respParameterData[tempPointer]) > LAcycCom_DriveValueFormats#FORMAT_DOUBLE_WORD) OR
                          ((TO_SINT(_respParameterData[tempPointer]) > LAcycCom_DriveValueFormats#FORMAT_FLOATING_POINT) AND (TO_SINT(_respParameterData[tempPointer]) < LAcycCom_DriveValueFormats#FORMAT_OCTET_STRING)) OR
                          ((TO_SINT(_respParameterData[tempPointer]) > LAcycCom_DriveValueFormats#FORMAT_OCTET_STRING) AND (TO_SINT(_respParameterData[tempPointer]) < LAcycCom_DriveValueFormats#FORMAT_TIME_DIFFERENCE)) OR
                          ((TO_SINT(_respParameterData[tempPointer]) > LAcycCom_DriveValueFormats#FORMAT_TIME_DIFFERENCE) AND (TO_SINT(_respParameterData[tempPointer]) < LAcycCom_DriveValueFormats#FORMAT_BYTE)) OR
                          (TO_SINT(_respParameterData[tempPointer]) < LAcycCom_DriveValueFormats#FORMAT_INTEGER_8))) AND (TO_SINT(_respParameterData[tempPointer]) <> LAcycCom_DriveValueFormats#FORMAT_ZERO)
                          THEN
                          // Format = Error, summarize the first and second error byte in a WORD error variable for each parameter
                          _parameter[tempIndex].errorValue := _respParameterData[tempPointer + 3];

                          // Points to the next parameter address
                          tempPointer := tempPointer + 6;

                          ELSE

                          CASE TO_SINT(_respParameterData[tempPointer]) OF
                              LAcycCom_DriveValueFormats#FORMAT_UNSIGNED_16:
                              tempWord.%B0 := _respParameterData[tempPointer + 3];
                              tempWord.%B1 := _respParameterData[tempPointer + 2];

                              _parameter[tempIndex].realValue := TO_REAL(TO_UINT(tempWord));
                              _parameter[tempIndex].errorValue := BYTE#16#FF; // Sets the error status and diagnostics
                              tempPointer := tempPointer + 4; // Points to the next parameter address

                              ELSE
                              // Wrong format. _parameter[n].format <> LAcycCom_DriveValueFormats#FORMAT_UNSIGNED_16
                              _firstParameterError := tempIndex;
                              diagnostics.firstParameterError := _firstParameterError;
                              _status := LAcycCom_DriveFunctionStatus#ERR_PARAMETER;
                              _error := TRUE;
                              _stateNumber := _fBSubState;
                              _fBState := LAcycCom_typeDriveActDeactStates#FB_ERROR;
                              EXIT;
                          END_CASE;

                          END_IF;

                      END_FOR;

                      IF (enableSavingOfWholeDriveSystem = FALSE) THEN // V1.5.3 "old" logic (save parameters of a specific DO) is active, i.e., if p971 is available, p971 is written, otherwise p977 is written if available (e.g. for drive S210)
                          IF (_parameter[0].errorValue = BYTE#16#FF) AND (_error = FALSE) THEN
                          // Write p971
                          _cmdBusy := FALSE;
                          _cmdError := FALSE;
                          _status := LAcycCom_DriveFunctionStatus#STATUS_BUSY;
                          _fBState := LAcycCom_typeDriveActDeactStates#FB_BUSY;
                          _fBSubState := LAcycCom_DriveRamToRomStates#FB_BUSY_WRITE_PARAM_971;
                          ELSIF (_parameter[1].errorValue = BYTE#16#FF)
                          AND (_error = FALSE)
                          THEN
                          // Write p977
                          _cmdBusy := FALSE;
                          _cmdError := FALSE;
                          _status := LAcycCom_DriveFunctionStatus#STATUS_BUSY;
                          _fBState := LAcycCom_typeDriveActDeactStates#FB_BUSY;
                          _fBSubState := LAcycCom_DriveRamToRomStates#FB_BUSY_WRITE_PARAM_977;
                          ELSIF (_parameter[0].errorValue = BYTE#16#19) AND (_parameter[1].errorValue = BYTE#16#19)
                          AND (_error = FALSE)
                          THEN
                          // 16#19 Drive object does not exist (access to a drive object that does not exist)
                          _firstParameterError := 0;
                          diagnostics.firstParameterError := _firstParameterError;
                          diagnostics.errorValue := _parameter[0].errorValue;
                          _status := LAcycCom_DriveFunctionStatus#ERR_DO_ID;
                          _error := TRUE;
                          _stateNumber := _fBSubState;
                          _fBState := LAcycCom_typeDriveActDeactStates#FB_ERROR;

                          ELSIF (_error = FALSE) THEN
                          // Both parameter are unavailable
                          _firstParameterError := 0;
                          diagnostics.firstParameterError := _firstParameterError;
                          diagnostics.errorValue := _parameter[0].errorValue;
                          _status := LAcycCom_DriveFunctionStatus#ERR_PARAMETER;
                          _error := TRUE;
                          _stateNumber := _fBSubState;
                          _fBState := LAcycCom_typeDriveActDeactStates#FB_ERROR;
                          END_IF;

                      ELSE // (enableSavingOfWholeDriveSystem = TRUE) V1.5.3 "new" logic to enable saving the parameters of the whole drive system is active, i.e., if p977 is available, p977 is written, otherwise p971 is written if available (e.g. for drive G120)
                          IF (_parameter[1].errorValue = BYTE#16#FF)
                          AND (_error = FALSE)
                          THEN
                          // Write p977
                          _cmdBusy := FALSE;
                          _cmdError := FALSE;
                          _status := LAcycCom_DriveFunctionStatus#STATUS_BUSY;
                          _fBState := LAcycCom_typeDriveActDeactStates#FB_BUSY;
                          _fBSubState := LAcycCom_DriveRamToRomStates#FB_BUSY_WRITE_PARAM_977;
                          ELSIF (_parameter[0].errorValue = BYTE#16#FF) AND (_error = FALSE) THEN
                          // Write p971
                          _cmdBusy := FALSE;
                          _cmdError := FALSE;
                          _status := LAcycCom_DriveFunctionStatus#STATUS_BUSY;
                          _fBState := LAcycCom_typeDriveActDeactStates#FB_BUSY;
                          _fBSubState := LAcycCom_DriveRamToRomStates#FB_BUSY_WRITE_PARAM_971;
                          ELSIF (_parameter[0].errorValue = BYTE#16#19) AND (_parameter[1].errorValue = BYTE#16#19)
                          AND (_error = FALSE)
                          THEN
                          // 16#19 Drive object does not exist (access to a drive object that does not exist)
                          _firstParameterError := 0;
                          diagnostics.firstParameterError := _firstParameterError;
                          diagnostics.errorValue := _parameter[0].errorValue;
                          _status := LAcycCom_DriveFunctionStatus#ERR_DO_ID;
                          _error := TRUE;
                          _stateNumber := _fBSubState;
                          _fBState := LAcycCom_typeDriveActDeactStates#FB_ERROR;

                          ELSIF (_error = FALSE) THEN
                          // Both parameter are unavailable
                          _firstParameterError := 0;
                          diagnostics.firstParameterError := _firstParameterError;
                          diagnostics.errorValue := _parameter[0].errorValue;
                          _status := LAcycCom_DriveFunctionStatus#ERR_PARAMETER;
                          _error := TRUE;
                          _stateNumber := _fBSubState;
                          _fBState := LAcycCom_typeDriveActDeactStates#FB_ERROR;
                          END_IF;
                      END_IF;

                      ELSIF (_fBSubState = LAcycCom_DriveRamToRomStates#FB_BUSY_ReadRecord_CHECK_971) OR (_fBSubState = LAcycCom_DriveRamToRomStates#FB_BUSY_ReadRecord_CHECK_977) THEN

                      _parameterRam2Rom[0].format := _respParameterData[0];  // Format of the parameter V1.3.3
                      // Format = Error
                      IF (((TO_SINT(_respParameterData[0]) > LAcycCom_DriveValueFormats#FORMAT_DOUBLE_WORD) OR
                          ((TO_SINT(_respParameterData[0]) > LAcycCom_DriveValueFormats#FORMAT_FLOATING_POINT) AND (TO_SINT(_respParameterData[0]) < LAcycCom_DriveValueFormats#FORMAT_OCTET_STRING)) OR
                          ((TO_SINT(_respParameterData[0]) > LAcycCom_DriveValueFormats#FORMAT_OCTET_STRING) AND (TO_SINT(_respParameterData[0]) < LAcycCom_DriveValueFormats#FORMAT_TIME_DIFFERENCE)) OR
                          ((TO_SINT(_respParameterData[0]) > LAcycCom_DriveValueFormats#FORMAT_TIME_DIFFERENCE) AND (TO_SINT(_respParameterData[0]) < LAcycCom_DriveValueFormats#FORMAT_BYTE)) OR
                          (TO_SINT(_respParameterData[0]) < LAcycCom_DriveValueFormats#FORMAT_INTEGER_8))) AND (TO_SINT(_respParameterData[0]) <> LAcycCom_DriveValueFormats#FORMAT_ZERO)
                      THEN
                          _parameterRam2Rom[0].errorValue := _respParameterData[3];
                          _firstParameterError := 0;
                          diagnostics.firstParameterError := _firstParameterError;
                          diagnostics.errorValue := _parameterRam2Rom[0].errorValue; // V1.3.2
                          _status := LAcycCom_DriveFunctionStatus#ERR_PARAMETER;

                          _error := TRUE;
                          _stateNumber := _fBSubState; // V1.3.2
                          _fBState := LAcycCom_typeDriveActDeactStates#FB_ERROR;

                      ELSE
                          // Analyse of the response buffer
                          CASE TO_SINT(_parameterRam2Rom[0].format) OF

                          LAcycCom_DriveValueFormats#FORMAT_UNSIGNED_16:
                              tempWord.%B0 := _respParameterData[3];
                              tempWord.%B1 := _respParameterData[2];
                              _parameterRam2Rom[0].realValue := TO_REAL(TO_UINT(tempWord));

                              _cmdBusy := FALSE;
                              _cmdError := FALSE;
                              _status := LAcycCom_DriveFunctionStatus#STATUS_BUSY;

                          ELSE
                              // Wrong format
                              _firstParameterError := 0;
                              diagnostics.firstParameterError := _firstParameterError;
                              _status := LAcycCom_DriveFunctionStatus#ERR_PARAMETER;
                              _error := TRUE;
                              _stateNumber := _fBSubState;
                              _fBState := LAcycCom_typeDriveActDeactStates#FB_ERROR;
                          END_CASE;

                          _parameterRam2Rom[0].errorValue := BYTE#16#FF; // Sets the error status and diagnostics

                      END_IF; // Format = Error

                      ELSE

                      // Error occurred during writing process (changing parameter values)
                      IF (_respParameterHeader.reqId = BYTE#16#82) THEN  // reqId: 16#82 (Error occurred during writing parameters)

                          _parameterRam2Rom[0].errorValue := _respParameterData[3];
                          // Save first parameter error in telegram
                          // V1.3.2
                          _firstParameterError := 0;
                          diagnostics.firstParameterError := _firstParameterError;
                          diagnostics.errorValue := _parameterRam2Rom[0].errorValue; // V1.3.2

                          _status := LAcycCom_DriveFunctionStatus#ERR_PARAMETER;
                          _error := TRUE;
                          _stateNumber := _fBSubState; // V1.3.2
                          _fBState := LAcycCom_typeDriveActDeactStates#FB_ERROR;

                      END_IF; // Error occurred during writing process (changing parameter values)
                      END_IF; // _cmdError = TRUE

                      IF (_fBSubState = LAcycCom_DriveRamToRomStates#FB_BUSY_ReadRecord_WRITE_PARAM_971) AND (_error = FALSE) THEN
                      _fBSubStateOld := LAcycCom_DriveRamToRomStates#FB_BUSY_CHECK_PARAM_971;
                      _fBSubState := LAcycCom_DriveRamToRomStates#FB_BUSY_CYCLE_TIMER;

                      ELSIF (_fBSubState = LAcycCom_DriveRamToRomStates#FB_BUSY_ReadRecord_CHECK_971) AND (_error = FALSE) THEN
                      _fBSubStateOld := LAcycCom_DriveRamToRomStates#FB_BUSY_CHECK_PARAM_971;
                      _fBSubState := LAcycCom_DriveRamToRomStates#FB_BUSY_CHECK_PROGRESS;

                      ELSIF (_fBSubState = LAcycCom_DriveRamToRomStates#FB_BUSY_ReadRecord_WRITE_PARAM_977) AND (_error = FALSE) THEN
                      _fBSubStateOld := LAcycCom_DriveRamToRomStates#FB_BUSY_CHECK_PARAM_977;
                      _fBSubState := LAcycCom_DriveRamToRomStates#FB_BUSY_CYCLE_TIMER;

                      ELSIF (_fBSubState = LAcycCom_DriveRamToRomStates#FB_BUSY_ReadRecord_CHECK_977) AND (_error = FALSE) THEN
                      _fBSubStateOld := LAcycCom_DriveRamToRomStates#FB_BUSY_CHECK_PARAM_977;
                      _fBSubState := LAcycCom_DriveRamToRomStates#FB_BUSY_CHECK_PROGRESS;

                      END_IF;
                  END_IF; // _cmdError = TRUE
                ELSE
                  _error := TRUE;
                  _stateNumber := _fbSubState;
                  _status := LAcycCom_DriveFunctionStatus#ERR_MISSMATCH_READ_BUFFER_SIZE;
                  _fbState := LAcycCom_typeDriveActDeactStates#FB_ERROR;
                END_IF;

                LAcycCom_DriveRamToRomStates#FB_BUSY_WAIT:
                // Timer for temporary errors
                _instOnDelay(signal := _timerStart,
                              duration := TIMER_TEMP_ERROR);

                _timerStart := TRUE;
                IF (_instOnDelay.output = TRUE) THEN
                    _timerStart := FALSE;
                    _fBSubState := _fBSubStateOld;
                END_IF;

                ELSE
                _error := TRUE;
                _status := LAcycCom_DriveFunctionStatus#ERR_UNDEFINED_SUBSTATE;
                _stateNumber := _fBSubState; // V1.3.2
                _fBState := LAcycCom_typeDriveActDeactStates#FB_ERROR;
            END_CASE;

            ELSE
            _error := TRUE;
            _status := LAcycCom_DriveFunctionStatus#ERR_COMMAND_TIMEOUT;
            _stateNumber := _fBSubState; // V1.3.2
            _fBState := LAcycCom_typeDriveActDeactStates#FB_ERROR;
            END_IF; // ((#buffer.element[_allocatedIndex].enable = TRUE) AND (_mode = #MODE_WITH_BUFFER_MANAGER)) OR _mode = #MODE_WITHOUT_BUFFER_MANAGER

            LAcycCom_typeDriveActDeactStates#FB_RELEASE:
            // Check buffer index for correctness
            IF (_allocatedIndex < 0) OR (_allocatedIndex > requestBufferHeader.bufferUpperBound) THEN
            _error := TRUE;
            _status := LAcycCom_DriveFunctionStatus#ERR_INVALID_BUF_INDEX;
            _stateNumber := _fBState;
            _fBState := LAcycCom_typeDriveActDeactStates#FB_ERROR;

            ELSIF (requestBufferHeader.lockBuffer = FALSE) THEN // V1.5.1
            requestBufferHeader.lockBuffer := TRUE;
            IF (requestBuffer[_allocatedIndex].state.%X0 = TRUE) THEN
                requestBuffer[_allocatedIndex].state.%X2 := TRUE;
            ELSE
                ;
            END_IF;
            requestBufferHeader.lockBuffer := FALSE;
            _status := LAcycCom_DriveFunctionStatus#STATUS_EXECUTION_FINISHED;
            _fBState := LAcycCom_typeDriveActDeactStates#FB_DONE;

            END_IF;

        ELSE
            _error := TRUE;
            _status := LAcycCom_DriveFunctionStatus#ERR_UNDEFINED_STATE;
            _stateNumber := _fBState;
            _fBState := LAcycCom_typeDriveActDeactStates#FB_ERROR;
        END_CASE;

        // If input execute is set during processing
        IF _warningRetriggering = TRUE AND _error = FALSE THEN
        _status := LAcycCom_DriveFunctionStatus#WARN_EXECUTE_SET_DURING_PROCESSING;
        END_IF;

    END_IF;

    //----------------------------------------------------------------------------------------------
    //Write outputs and error handling
    //----------------------------------------------------------------------------------------------

    // Error occurred in request
    IF (_fBState = LAcycCom_typeDriveActDeactStates#FB_ERROR) THEN

        // Release the allocated element when error occurs
        IF (_stateNumber <> LAcycCom_typeDriveActDeactStates#FB_FIRST_CYCLE) AND (_stateNumber <> LAcycCom_typeDriveActDeactStates#FB_ALLOCATE)
        AND (_busy = TRUE) AND (_withoutResourceManager = FALSE)
        THEN
        IF requestBufferHeader.lockBuffer = FALSE THEN  // V1.5.1
            requestBufferHeader.lockBuffer := TRUE;
            IF (requestBuffer[_allocatedIndex].state.%X0 = TRUE) THEN
            requestBuffer[_allocatedIndex].state.%X2 := TRUE;
            ELSE
            ;
            END_IF;
            requestBufferHeader.lockBuffer := FALSE;

            // Write diagnostics
            diagnostics.stateNumber := _stateNumber;
            diagnostics.subfunctionStatus := _subfunctionStatus;
            diagnostics.status := _status;
            _busy := FALSE;
            _done := FALSE;

        END_IF;

        ELSE
        // Write diagnostics
        diagnostics.stateNumber := _stateNumber;
        diagnostics.subfunctionStatus := _subfunctionStatus;
        diagnostics.status := _status;
        _busy := FALSE;
        _done := FALSE;
        END_IF;

        // Request finished
    ELSIF (_fBState = LAcycCom_typeDriveActDeactStates#FB_DONE) THEN

        // Output for one cycle minimum
        IF (execute = FALSE) AND (_done = TRUE) THEN
        _done := FALSE;
        _status := LAcycCom_DriveFunctionStatus#STATUS_NO_CALL;
        _fBState := LAcycCom_typeDriveActDeactStates#FB_IDLE;

        ELSE
        _done := TRUE;
        _busy := FALSE;
        END_IF;
        // If input execute is set during processing
        IF _warningRetriggering = TRUE THEN
        _status := LAcycCom_DriveFunctionStatus#ERR_AMBIGUOUS_FB_CALL;
        diagnostics.status := _status;
        _error := TRUE;
        _done := FALSE;
        END_IF;
    END_IF;

    // Write static values to outputs
    IF _busy = FALSE OR _error = FALSE
    THEN  // V1.5.1
        error := _error;
        status := _status;
    END_IF;
    busy := _busy;
    done := _done;
  END_FUNCTION_BLOCK
END_NAMESPACE

(* ---- LAcycCom_ReadDriveMessagesDateTime.st ---- *)
USING System.Timer;
USING System.DateTime;
USING Siemens.Simatic.Hardware.Utilities;
USING Siemens.Simatic.Clocks;

NAMESPACE Simatic.Ax.LAcycCom.Procedural
  TYPE
    LAcycCom_ReadDriveMessagesDateTimeStates : SINT (
      FB_IDLE := SINT#0,   // Idle state in FB
      FB_ALARMS_DATASET := SINT#1,   // Preparing dataset state in FB (alarms)
      FB_FAULTS_DATASET := SINT#2,   // Preparing dataset state in FB (faults)
      FB_SIMESSAGES_DATASET := SINT#3,   // Preparing dataset state in FB (SI messages )
      FB_ALARMS_GONE_DATASET := SINT#4,   // State that prepare dataset (r2125) and call ReadDriveParams
      FB_READ_STEP_1 := SINT#5,   // Call ReadDriveParams and write messages in statBuffer state
      FB_READ_STEP_2 := SINT#6,   // Call ReadDriveParams with FALSE state
      FB_SORTING := SINT#10   // Sorting state in FB
    ) := FB_IDLE;
  END_TYPE

  ///-----------------------------------------------------------------------------
	/// SIEMENS AG
	/// (c)Copyright 2026 All Rights Reserved
	///-----------------------------------------------------------------------------
	/// Library: LAcycCom
	/// Tested with: S7-1513-1 PN
	/// Engineering: SIMATIC AX
	/// Restrictions: The drive must be in UTC mode
	/// Requirements: S7-1200 / S7-1500
	///               FB LAcycCom_ResourceManager is required
	/// Functionality: Read alarms, faults and SI messages from SINAMICS drive and
	///                output in structure (newest elements first)
  ///-----------------------------------------------------------------------------
  FUNCTION_BLOCK LAcycCom_ReadDriveMessagesDateTime
    {S7.Extern = ReadWrite}
    VAR_INPUT
      execute : BOOL;   /// TRUE: Rising edge starts the functionality once
      alarms : BOOL := TRUE;   /// TRUE: Enable reading of alarms
      faults : BOOL := TRUE;   /// TRUE: Enable reading of faults
      siMessages : BOOL;   /// TRUE: Enable reading of SI messages
      driveObjectId : INT := -1;   /// Optional: Identification number of the drive object (value <0: driveObjectId is not used, i.e. the corresponding drive object is only addressed via the hardwareId)
      hardwareId : UINT;   /// Hardware identifier of the hardware module
    END_VAR

    {S7.Extern = ReadOnly}
    VAR_OUTPUT
      done : BOOL;   /// TRUE: Commanded action has been completed successfully
      busy : BOOL;   /// TRUE: FB is not finished and new output values can be expected
      error : BOOL;   /// TRUE: Rising edge informs that an error occurred during the execution of the FB
      status : LAcycCom_DriveFunctionStatus;   /// Status identifier
      diagnostics : LAcycCom_typeDriveDiagnostics;   /// Diagnostics structure
      messages : ARRAY[0..MESSAGES_COUNT_UPPER_LIM] OF LAcycCom_typeDriveMessage;   /// List of drive messages
    END_VAR

    VAR_IN_OUT
      requestBufferHeader : LAcycCom_typeRequestBufferHeader;   /// Interface for header of request buffer
      requestBuffer : ARRAY[*] OF LAcycCom_typeRequestBufferElement;   /// Interface for request buffer
    END_VAR

    VAR
      _busy : BOOL;   /// Static value for output busy
      _done : BOOL;   /// Static value for output done
      _error : BOOL;   /// Static value for output error
      _status : LAcycCom_DriveFunctionStatus;   /// Static value for output status
      _executeOld : BOOL;   /// Old value of execute for edge detection
      _fbState : LAcycCom_ReadDriveMessagesDateTimeStates;   /// States in the function block state machine
      _alarmsInput : BOOL;   /// Static variable for input "alarms"
      _faultsInput : BOOL;   /// Static variable for input "faults"
      _siMessagesInput : BOOL;   /// Static variable for input "siMessages"
      _driveObjectId : INT;   /// Intern identification number of the drive object
      _hardwareId : UINT;   /// Intern hardware identifier of the hardware module
      _dtl : LDATE_AND_TIME;   /// Time varible for comparasion (sorting)
      _indexNew : DINT;   /// Index of newest elemet (for sorting)
      _offset : SINT;   /// Offset for statBuffer/ first empty element in statBuffer
      _warningNoMessages : BOOL;   /// TRUE: At least one of three inputs must be selected
      _warningRetriggering : BOOL;   /// TRUE: Input execute is set during processing
      _faultsComplete : BOOL;   /// TRUE: FB_READ state complete successfully (faults)
      _alarmsComplete : BOOL;   /// TRUE: FB_READ state complete successfully (alarms)
      _currentMessage : SINT;   /// Static variable represents current message type
      _goneAlarms : ARRAY[0..ELEMENTS_COUNT_UPPER_LIM] OF BOOL;   /// TRUE: this alarm is already gone
      _dataset : ARRAY[0..PARAMETER_COUNT_READ_UPPER_LIM] OF LAcycCom_typeDriveDataset;   /// Dataset for LAcycCom_ReadDriveParams
      _buffer : ARRAY[0..MESSAGES_COUNT_UPPER_LIM] OF LAcycCom_typeDriveMessage;   /// Buffer for store alarms, faults and SI messages
      _instReadDriveParams : LAcycCom_ReadDriveParams;   /// Instance of LAcycCom_ReadDriveParams
    END_VAR

    VAR_TEMP
      tempIndex : DINT;   // Temporary loop index variable
      tempSort : SINT;   // Temporary loop variable for sorting
      tempUInt : UInt;   // Temporary UInt variable
      tempDate : LDATE;   // Temporary variable for date
      tempTime : LTIME_OF_DAY;   // Temporary variable for time
      tempRetValWord : WORD;   // Return value of system function as word
      tempDTL : LDATE_AND_TIME;   // Temporary DTL variable
      tempGeoAddr : GeoAddr;   // Current Geo Address information
      tempVoidDiagnostics : LAcycCom_typeDriveDiagnostics;   // Temporary empty diagnostics structure
      tempVoidMessage : LAcycCom_typeDriveMessage;   // Temporary empty message structure
    END_VAR

    VAR CONSTANT
      INT_ERR_NOT_CONFIG : WORD := WORD#16#8093;   // The DP component addressed via ID or F_ID is not configured (ReadRecord/WriteRecord)
      INT_ERR_NOT_KNOWN : WORD := WORD#16#80B0;   // Data record not known in module. Illegal data record number ≥ 256 (ReadRecord/WriteRecord)
      INT_ERR_LOG_START_ADDR : WORD := WORD#16#8090;   // Invalid logical start address (ReadRecord/WriteRecord)
      DO_NOT_EXIST : WORD := WORD#16#0019;   // Drive object does not exist
      OFFSET_INFO : SINT := SINT#8;   // Offset in dataset for "info" information
      OFFSET_DAYS : SINT := SINT#16;   // Offset in dataset for "Count days" information
      OFFSET_MS : SINT := SINT#24;   // Offset in dataset for "Count ms" information
      PARAMETER_COUNT_READ_UPPER_LIM : INT := 31;   // Count of parameters to be read in ReadDriveParams
      ELEMENTS_COUNT_UPPER_LIM : INT := 7;   // Count of elements in one message type
      MAX_DRIVE_OBJECT_NO : INT := 254;   // Maximum drive object number limited by SINAMICS p101
      MESSAGES_COUNT_UPPER_LIM : INT := 23;   // Maxmimum number of messages
      DAYS_TO_NS : LREAL := LREAL#1.0e+9 * 3600 * 24;   // Conversion value for days to ns
    END_VAR

    // Check if FB is triggered
    IF (execute = TRUE) AND (_executeOld = FALSE) AND (_busy = TRUE) THEN
      // Input execute is set during processing
      status := LAcycCom_DriveFunctionStatus#WARN_EXECUTE_SET_DURING_PROCESSING;
      _warningRetriggering := TRUE;
      _executeOld := execute;

    ELSIF (execute = TRUE) AND (_executeOld = FALSE) THEN
      // First call
      // Functionality is busy
      _busy := TRUE;

      // Reset other outputs
      _error := FALSE;
      _done := FALSE;
      _status := LAcycCom_DriveFunctionStatus#STATUS_FIRST_CALL;
      status := _status;

      busy := _busy;
      error := _error;
      done := _done;
      _executeOld := execute;

      // Initialize
      _alarmsInput := alarms;
      _faultsInput := faults;
      _siMessagesInput := siMessages;
      _driveObjectId := driveObjectId;
      _hardwareId := hardwareId;
      _offset := SINT#0;
      _indexNew := 0;
      diagnostics := tempVoidDiagnostics;
      diagnostics.firstParameterError := -1; // V1.3.2
      diagnostics.errorValue := BYTE#16#FF; // V1.3.2
      _warningNoMessages := FALSE;
      _warningRetriggering := FALSE;
      _currentMessage := SINT#0;
      _faultsComplete := FALSE;
      _alarmsComplete := FALSE;
      // Set a default value to first entry in dataset
      _dataset[0].errorValue := BYTE#16#FF;
      // Set init time for comparison (sorting)
      _dtl := tempDTL;

      IF (_driveObjectId > MAX_DRIVE_OBJECT_NO)
        OR (_driveObjectId = 0)
      THEN // V1.5.2
        // Wrong drive object ID at input
        _error := TRUE;
        _status := LAcycCom_DriveFunctionStatus#ERR_INVALID_DRIVE_OBJECT_ID;
        RETURN;
      END_IF;

      // Clearing static and output area for alarms, faults and SI messages
      FOR tempIndex := 0 TO MESSAGES_COUNT_UPPER_LIM DO
        _buffer[tempIndex] := tempVoidMessage;
      END_FOR;

      // Write diagnostics
      diagnostics.hardwareId := _hardwareId;

      // Call ReadDriveParams with FALSE
      _instReadDriveParams(execute := FALSE,
                          requestBufferHeader := requestBufferHeader,
                          requestBuffer := requestBuffer,
                          dataset := _dataset);

      // Check if device hardware address exist
      tempRetValWord := ReadSlotFromHardwareID(hardwareId := _hardwareId,
                                               geoAddr := tempGeoAddr);

      // Check if everything is okay
      IF tempRetValWord <> WORD#16#0 THEN
        _error := TRUE;
        diagnostics.subfunctionStatus := tempRetValWord;
        _status := LAcycCom_DriveFunctionStatus#ERR_GET_LOCAL_DATE_TIME;
        RETURN;
      END_IF;

      // Alarms or faults or SI messages
      IF _siMessagesInput = TRUE THEN
        _fbState := LAcycCom_ReadDriveMessagesDateTimeStates#FB_SIMESSAGES_DATASET;
      ELSIF _faultsInput = TRUE THEN
        _fbState := LAcycCom_ReadDriveMessagesDateTimeStates#FB_FAULTS_DATASET;
      ELSIF _alarmsInput = TRUE THEN
        _fbState := LAcycCom_ReadDriveMessagesDateTimeStates#FB_ALARMS_GONE_DATASET;
      ELSE
        // Warning. At least one of three inputs must be selected
        _status := LAcycCom_DriveFunctionStatus#STATUS_FINISHED_NO_MSG_SELECTED;
        _fbState := LAcycCom_ReadDriveMessagesDateTimeStates#FB_SORTING;
        _warningNoMessages := TRUE;
      END_IF;
      RETURN;

      // Check if FB is disabled (falling edge) after job is done or FB is in error state
    ELSIF (execute = FALSE AND _busy = FALSE) AND
      (_error = TRUE OR _done = TRUE)
    THEN
      // Error outputs are reset with falling edge of enable input
      _error := FALSE;

      // Enable and busy are reset with falling edge of enable input
      _done := FALSE;
      _busy := FALSE;

      // Write outputs
      _status := LAcycCom_DriveFunctionStatus#STATUS_NO_CALL;
      status := _status;
      busy := _busy;
      done := _done;
      error := _error;
      _fbState := LAcycCom_ReadDriveMessagesDateTimeStates#FB_IDLE;

      // Clearing static and output area for alarms, faults and SI messages
      FOR tempIndex := 0 TO MESSAGES_COUNT_UPPER_LIM DO
        _buffer[tempIndex] := tempVoidMessage;
      END_FOR;

      _executeOld := execute;
      RETURN;

      // FB is currently executed and not finished
    ELSIF _busy = TRUE THEN
      _executeOld := execute;

      // FB is disabled
    ELSE
      _executeOld := execute;
      RETURN;
    END_IF;

    //----------------------------------------------------------------------------------------------
    IF (_busy = TRUE) AND (_error = FALSE) THEN  // Functionality running
      CASE _fbState OF
        LAcycCom_ReadDriveMessagesDateTimeStates#FB_ALARMS_DATASET:
          // Preparing dataset for ReadDriveParams
          // Alarms
          FOR tempIndex := 0 TO ELEMENTS_COUNT_UPPER_LIM DO
            tempUInt := TO_UINT(tempIndex);
            // Index 0 ..7 - r2122 - "Alarm Code"
            _dataset[tempIndex].parameterNumber := UINT#2122;
            _dataset[tempIndex].index := tempUInt;
            // Index 8 ..15 - r2124 - "Alarm Info"
            _dataset[tempIndex + OFFSET_INFO].parameterNumber := UINT#2124;
            _dataset[tempIndex + OFFSET_INFO].index := tempUInt;
            // Index 16 .. 23 - r2145 - "Alarm come time in days"
            _dataset[tempIndex + OFFSET_DAYS].parameterNumber := UINT#2145;
            _dataset[tempIndex + OFFSET_DAYS].index := tempUInt;
            // Index 24 .. 31 - r2123 - "Alarm come time in ms"
            _dataset[tempIndex + OFFSET_MS].parameterNumber := UINT#2123;
            _dataset[tempIndex + OFFSET_MS].index := tempUInt;
          END_FOR;
          _fbState := LAcycCom_ReadDriveMessagesDateTimeStates#FB_READ_STEP_1;
          _currentMessage := LAcycCom_DriveMessageType#ALARM;

        LAcycCom_ReadDriveMessagesDateTimeStates#FB_FAULTS_DATASET:
          // Preparing dataset for ReadDriveParams
          // Faults
          FOR tempIndex := 0 TO ELEMENTS_COUNT_UPPER_LIM DO
            tempUInt := TO_UINT(tempIndex);
            // Index 0 ..7 - r945 - "Fault Code"
            _dataset[tempIndex].parameterNumber := UINT#945;
            _dataset[tempIndex].index := tempUInt;
            // Index 8 ..15 - r949 - "Fault Info"
            _dataset[tempIndex + OFFSET_INFO].parameterNumber := UINT#949;
            _dataset[tempIndex + OFFSET_INFO].index := tempUInt;
            // Index 16 .. 23 - r2130 - "Fault come time in days"
            _dataset[tempIndex + OFFSET_DAYS].parameterNumber := UINT#2130;
            _dataset[tempIndex + OFFSET_DAYS].index := tempUInt;
            // Index 24 .. 31 - r948 - "Fault come time in ms"
            _dataset[tempIndex + OFFSET_MS].parameterNumber := UINT#948;
            _dataset[tempIndex + OFFSET_MS].index := tempUInt;
            _goneAlarms[tempIndex] := FALSE;
          END_FOR;
          _fbState := LAcycCom_ReadDriveMessagesDateTimeStates#FB_READ_STEP_1;
          _currentMessage := LAcycCom_DriveMessageType#FAULT;

        LAcycCom_ReadDriveMessagesDateTimeStates#FB_SIMESSAGES_DATASET:
          // Preparing dataset for ReadDriveParams
          // SI Messages
          FOR tempIndex := 0 TO ELEMENTS_COUNT_UPPER_LIM DO
            tempUInt := TO_UINT(tempIndex);
            // Index 0 ..7 - r9747 - "SI Code"
            _dataset[tempIndex].parameterNumber := UINT#9747;
            _dataset[tempIndex].index := tempUInt;
            // Index 8 ..15 - r9749 - "SI Info"
            _dataset[tempIndex + OFFSET_INFO].parameterNumber := UINT#9749;
            _dataset[tempIndex + OFFSET_INFO].index := tempUInt;
            // Index 16 .. 23 - r9754- "SI Message come time in days"
            _dataset[tempIndex + OFFSET_DAYS].parameterNumber := UINT#9754;
            _dataset[tempIndex + OFFSET_DAYS].index := tempUInt;
            // Index 24 .. 31 - r9748 - "SI Message come time in ms"
            _dataset[tempIndex + OFFSET_MS].parameterNumber := UINT#9748;
            _dataset[tempIndex + OFFSET_MS].index := tempUInt;
            _goneAlarms[tempIndex] := FALSE;
          END_FOR;
          _fbState := LAcycCom_ReadDriveMessagesDateTimeStates#FB_READ_STEP_1;
          _currentMessage := LAcycCom_DriveMessageType#SI_MESSAGE;

        LAcycCom_ReadDriveMessagesDateTimeStates#FB_ALARMS_GONE_DATASET:
          IF NOT _instReadDriveParams.busy AND
            NOT _instReadDriveParams.done AND
            NOT _instReadDriveParams.error
          THEN
            // Prepare dataset
            FOR tempIndex := 0 TO ELEMENTS_COUNT_UPPER_LIM DO
              tempUInt := TO_UINT(tempIndex);
              // Index 0..7 - r2125 - "Alarm time removed in milliseconds"
              _dataset[tempIndex].parameterNumber := UINT#2125;
              _dataset[tempIndex].index := tempUInt;
            END_FOR;
          END_IF;

          // Call ReadDriveParams
          _instReadDriveParams(execute := TRUE,
                              parameterCount := ELEMENTS_COUNT_UPPER_LIM + 1, // 8 parameter
                              driveObjectId := _driveObjectId,
                              hardwareId := _hardwareId,
                              requestBufferHeader := requestBufferHeader,
                              requestBuffer := requestBuffer,
                              dataset := _dataset);

          IF NOT _instReadDriveParams.busy THEN
            diagnostics := _instReadDriveParams.diagnostics;
            IF _instReadDriveParams.done = TRUE THEN
              // To determine what alarms are already gone
              FOR tempIndex := 0 TO ELEMENTS_COUNT_UPPER_LIM DO
                IF _dataset[tempIndex].dwordValue <> DWORD#16#0 THEN
                  _goneAlarms[tempIndex] := TRUE;
                ELSE
                  _goneAlarms[tempIndex] := FALSE; // 01.05.03
                END_IF;
              END_FOR;

              // Call ReadDriveParams with FALSE
              _instReadDriveParams(execute := FALSE,
                                  requestBufferHeader := requestBufferHeader,
                                  requestBuffer := requestBuffer,
                                  dataset := _dataset);
              // Go next
              _fbState := LAcycCom_ReadDriveMessagesDateTimeStates#FB_ALARMS_DATASET;

            ELSIF _instReadDriveParams.error = TRUE THEN
              _error := TRUE;
              // HwId is wrong
              IF (_instReadDriveParams.status = LAcycCom_DriveFunctionStatus#ERR_WRITERECORD OR _instReadDriveParams.status = LAcycCom_DriveFunctionStatus#ERR_READRECORD) AND
                ((_instReadDriveParams.diagnostics.subfunctionStatus = INT_ERR_NOT_CONFIG)
                OR (_instReadDriveParams.diagnostics.subfunctionStatus = INT_ERR_NOT_KNOWN)
                OR (_instReadDriveParams.diagnostics.subfunctionStatus = INT_ERR_LOG_START_ADDR))
              THEN
                _status := LAcycCom_DriveFunctionStatus#ERR_HW_ID;
                // Drive object does not exist
              ELSIF _dataset[0].errorValue = DO_NOT_EXIST THEN
                _status := LAcycCom_DriveFunctionStatus#ERR_DO_ID;
              ELSE
                _status := LAcycCom_DriveFunctionStatus#ERR_READ_DRIVE_PARAMS_ALARMS_GONE;
              END_IF;
            END_IF;
          END_IF;

          LAcycCom_ReadDriveMessagesDateTimeStates#FB_READ_STEP_1:
          // Call ReadDriveParams
          _instReadDriveParams(execute := TRUE,
                              parameterCount := PARAMETER_COUNT_READ_UPPER_LIM + 1, // 32 parameter
                              driveObjectId := _driveObjectId,
                              hardwareId := _hardwareId,
                              requestBufferHeader := requestBufferHeader,
                              requestBuffer := requestBuffer,
                              dataset := _dataset);

          IF NOT _instReadDriveParams.busy THEN
            diagnostics := _instReadDriveParams.diagnostics;
            IF _instReadDriveParams.done = TRUE THEN
              // Copy to static area only elements with content
              FOR tempIndex := 0 TO ELEMENTS_COUNT_UPPER_LIM DO
                IF NOT _goneAlarms[tempIndex] THEN
                  _buffer[_offset].code := TO_UINT(_dataset[tempIndex].dwordValue);
                  // If parameter empty - then go next
                  IF _dataset[tempIndex].dwordValue = WORD#16#0 THEN
                    EXIT;
                  END_IF;
                  _buffer[_offset].messageType := _currentMessage; // Identifier for message
                  _buffer[_offset].info := TO_UDINT(_dataset[tempIndex + OFFSET_INFO].dwordValue);
                  tempDate := TO_LDATE(TO_LWORD(TO_LINT(_dataset[tempIndex + OFFSET_DAYS].dwordValue) * TO_LINT(DAYS_TO_NS)));
                  tempTime := TO_LTOD(TO_LWORD(TO_LINT(_dataset[tempIndex + OFFSET_MS].dwordValue) * LINT#1000000));
                  NewDateAndTime(tempDate, tempTime, _buffer[_offset].comeDateAndTime); // generate LDT format from LDATE and LTIME_OF_DAY
                  _offset := _offset + SINT#1;
                END_IF;
              END_FOR;
              // Set "complete" flag
              CASE _currentMessage OF
                LAcycCom_DriveMessageType#ALARM:
                  _alarmsComplete := TRUE;
                LAcycCom_DriveMessageType#FAULT:
                  _faultsComplete := TRUE;
                ELSE
                  ;
              END_CASE;
              // Go next step
              _fbState := LAcycCom_ReadDriveMessagesDateTimeStates#FB_READ_STEP_2;

              // Error while reading  with ReadDriveParams
            ELSIF _instReadDriveParams.error = TRUE THEN
              _error := TRUE;
              // HwId is wrong
              IF (_instReadDriveParams.status = LAcycCom_DriveFunctionStatus#ERR_WRITERECORD OR _instReadDriveParams.status = LAcycCom_DriveFunctionStatus#ERR_READRECORD) AND
                ((_instReadDriveParams.diagnostics.subfunctionStatus = INT_ERR_NOT_CONFIG)
                OR (_instReadDriveParams.diagnostics.subfunctionStatus = INT_ERR_NOT_KNOWN)
                OR (_instReadDriveParams.diagnostics.subfunctionStatus = INT_ERR_LOG_START_ADDR))
              THEN
                _status := LAcycCom_DriveFunctionStatus#ERR_HW_ID;
                // Drive object does not exist
              ELSIF _dataset[0].errorValue = DO_NOT_EXIST THEN
                _status := LAcycCom_DriveFunctionStatus#ERR_DO_ID;
              ELSE
                CASE _currentMessage OF
                  LAcycCom_DriveMessageType#ALARM:
                    _status := LAcycCom_DriveFunctionStatus#ERR_READ_DRIVE_PARAMS_ALARMS;
                    LAcycCom_DriveMessageType#FAULT:
                    _status := LAcycCom_DriveFunctionStatus#ERR_READ_DRIVE_PARAMS_FAULTS;
                    LAcycCom_DriveMessageType#SI_MESSAGE:
                    _status := LAcycCom_DriveFunctionStatus#ERR_READ_DRIVE_PARAMS_SI_MESSAGES;
                  ELSE
                    ;
                END_CASE;
              END_IF;
            END_IF;
          END_IF;

        LAcycCom_ReadDriveMessagesDateTimeStates#FB_READ_STEP_2:
          // Call ReadDriveParams with FALSE
          _instReadDriveParams(execute := FALSE,
                              requestBufferHeader := requestBufferHeader,
                              requestBuffer := requestBuffer,
                              dataset := _dataset);

          // Choice next step. Right call order: SI messages, faults, alarms
          IF _faultsInput AND NOT _faultsComplete THEN
            _fbState := LAcycCom_ReadDriveMessagesDateTimeStates#FB_FAULTS_DATASET;
          ELSIF (_alarmsInput AND NOT _alarmsComplete) THEN
            _fbState := LAcycCom_ReadDriveMessagesDateTimeStates#FB_ALARMS_GONE_DATASET;
          ELSE
            _fbState := LAcycCom_ReadDriveMessagesDateTimeStates#FB_SORTING;
          END_IF;

        LAcycCom_ReadDriveMessagesDateTimeStates#FB_SORTING:
          // When at least one message has been read
          IF _offset <> 0 THEN
            // Sorting algorithm. Newest message - first
            // When more then two messages of different type have the same come time, then order sequence is - alarms, faults, SI messages
            FOR tempSort := 0 TO (_offset - SINT#1) DO
              // Find newest element
              FOR tempIndex := 0 TO (_offset - 1) DO
                IF _buffer[tempIndex].comeDateAndTime >= _dtl THEN
                  _dtl := _buffer[tempIndex].comeDateAndTime;
                  _indexNew := tempIndex;
                END_IF;
              END_FOR;

              // Copy found element to output structure
              messages[tempSort] := _buffer[_indexNew];

              // Remove this element from buffer - by setting the value as small as possible
              _buffer[_indexNew].comeDateAndTime := tempDTL;
              // Set init time for next comparison
              _dtl := tempDTL;
            END_FOR;
          END_IF;
          // Set "done" flag
          _done := TRUE;

        ELSE
          _error := TRUE;
          _status := LAcycCom_DriveFunctionStatus#ERR_UNDEFINED_STATE;
      END_CASE;
    END_IF;

    //----------------------------------------------------------------------------------------------
    // Write outputs and error handling
    //----------------------------------------------------------------------------------------------
    // Error occurred in request
    IF _error = TRUE
    THEN
      _done := FALSE;
      _busy := FALSE;
      // Write diagnostics
      diagnostics.stateNumber := _fbState;
      diagnostics.status := _status;

      // Request finished
    ELSIF _done = TRUE
    THEN
      _busy := FALSE;
      _error := FALSE;
      _fbState := LAcycCom_ReadDriveMessagesDateTimeStates#FB_IDLE;
      // Set status
      IF _warningRetriggering = TRUE THEN
        // If input execute is set during processing
        _status := LAcycCom_DriveFunctionStatus#ERR_AMBIGUOUS_FB_CALL;
        diagnostics.status := _status;
        _error := TRUE;
        _done := FALSE;
      ELSIF _warningNoMessages = FALSE THEN
        // Execution finished without errors
        _status := LAcycCom_DriveFunctionStatus#STATUS_EXECUTION_FINISHED;
      ELSE
        // Warning. At least one of three inputs must be selected
        _status := LAcycCom_DriveFunctionStatus#STATUS_FINISHED_NO_MSG_SELECTED;
        diagnostics.status := _status;
      END_IF;

      // If input execute is set during processing
    ELSIF _warningRetriggering = TRUE
    THEN
      _status := LAcycCom_DriveFunctionStatus#WARN_EXECUTE_SET_DURING_PROCESSING;

      // Request in execution
    ELSE
      _status := LAcycCom_DriveFunctionStatus#STATUS_SUBSEQUENT_CALL;
    END_IF;

    // Write static values to outputs
    done := _done;
    busy := _busy;
    error := _error;
    status := _status;
    //----------------------------------------------------------------------------------------------
  END_FUNCTION_BLOCK
END_NAMESPACE
